// TwinCAT 3 PLC project PeerToPeerB
// ProgramVersion: 3.1.0.5
// libraries:
//   Tc2_Standard, * (Beckhoff Automation GmbH)
//   Tc2_System, * (Beckhoff Automation GmbH)
//   Tc2_TcpIp, * (Beckhoff Automation GmbH)
//   Tc2_Utilities, * (Beckhoff Automation GmbH)
//   Tc3_Module, * (Beckhoff Automation GmbH)
// project tree:
//   Data types/ E_ClientServerSteps.TcDUT, ST_FrameFifoEntry.TcDUT
//   Global Variables/ Global_Variables.TcGVL
//   POUs/ FB_PeerToPeer.TcPOU, MAIN.TcPOU
//   POUs/Helper POUs/ FB_FrameFifo.TcPOU, FB_LogFifo.TcPOU
//   / StandardB.TcTTO
// real-time tasks:
//   TASK StandardB: cycle T#10ms, priority 21, ADS port 351

CONFIGURATION PeerToPeerB
    RESOURCE PLC ON TwinCAT3
        TASK StandardB(INTERVAL := T#10ms, PRIORITY := 21);
        PROGRAM MAIN WITH StandardB : MAIN;
    END_RESOURCE
END_CONFIGURATION

// ---- Data types/E_ClientServerSteps.TcDUT
TYPE E_ClientServerSteps :
(
	eUDP_STATE_IDLE		:= 0,
	eUDP_STATE_CREATE_START,
	eUDP_STATE_CREATE_WAIT,
	eUDP_STATE_SEND_START,
	eUDP_STATE_SEND_WAIT,
	eUDP_STATE_RECEIVE_START,
	eUDP_STATE_RECEIVE_WAIT,
	eUDP_STATE_CLOSE_START,
	eUDP_STATE_CLOSE_WAIT,
	eUDP_STATE_ERROR
);
END_TYPE

// ---- Data types/ST_FrameFifoEntry.TcDUT
TYPE ST_FrameFifoEntry :
STRUCT
	stRemoteAddr 	: ST_SockAddr;(* Remote address. String containing an (Ipv4) Internet Protocol dotted address and port number. *)
	sMessage		: T_MaxString;	(* UDP packet data *)
END_STRUCT
END_TYPE

// ---- Global Variables/Global_Variables.TcGVL
VAR_GLOBAL CONSTANT
	PLCPRJ_BUFFER_SIZE					: UDINT := 1000;(* Max. internal fifo/receiver buffer size *)

	(* Some project specific error codes *)
	PLCPRJ_ERROR_SENDFIFO_OVERFLOW		: UDINT := 16#8103;
	PLCPRJ_ERROR_RECFIFO_OVERFLOW		: UDINT := 16#8104;
END_VAR

// ---- POUs/MAIN.TcPOU
PROGRAM MAIN
VAR
	bSendOnceToItself	: BOOL;(* Rising edge at this variable sends message to local host/port (itself) *)
	bSendOnceToRemote	: BOOL;(* Rising edge at this variable sends message to the remote host/port *)
	sSrvNetId			: T_AmsNetID 	:= '';(* TwinCAT TCP/IP server network address. Default: empty string. *)
	sLocalHost			: T_IPv4Addr 	:= '127.0.0.1';(* Local address: String containing an (Ipv4) Internet Protocol dotted address. *) 
	nLocalPort			: UDINT			:= 11000;(* Local address: IP port number *)
	sRemoteHost			: T_IPv4Addr 	:= '127.0.0.1';(* Remote address: String containing an (Ipv4) Internet Protocol dotted address. *)
	nRemotePort			: UDINT 		:= 10000;(* Remote address: IP port number. *)
	bEnable				: BOOL 			:= TRUE;(* TRUE => Enable/connect, FALSE => Disable/disconnect *)
	bLog				: BOOL			:= TRUE;(* TRUE => Enable log message output, FALSE => Disable *)
	
	fbPeerToPeer		: FB_PeerToPeer := ( sPrefix := 'PeerToPeerB::' ) ;
	
   	fbTx				: FB_FrameFifo;
   	fbRx				: FB_FrameFifo;
   	fbLog				: FB_LogFifo;
	
   	stSendTo			: ST_FrameFifoEntry;
   	stReceivedFrom		: ST_FrameFifoEntry;
	sLoggedMessage		: T_MaxString;

   	fbCloseAll 			: FB_SocketCloseAll;
   	bInitialize			: BOOL := TRUE;
END_VAR

(* On PLC reset or program download close all opened/created sockets *)
fbCloseAll( sSrvNetId := sSrvNetId, bExecute:= bInitialize );
IF fbCloseAll.bBusy OR fbCloseAll.bError THEN
	RETURN;
END_IF
bInitialize := FALSE;

(* Send and receive messages *)
fbPeerToPeer( 	sSrvNetId := sSrvNetId, 
				fbTx := fbTx, 
				fbRx := fbRx,
				fbLog := fbLog, 
				sLocalHost := sLocalHost, 
				nLocalPort := nLocalPort, 
				bEnable := bEnable, bLog := bLog );

IF fbPeerToPeer.bCreated THEN
	
	IF bSendOnceToRemote THEN
		bSendOnceToRemote 			:= FALSE;		(* Clear flag *)
		stSendTo.stRemoteAddr.sAddr := sRemoteHost;	(* Remote host IP address *)
		stSendTo.stRemoteAddr.nPort := nRemotePort;	(* Remote host port number *)
		stSendTo.sMessage			:= 'Hello remote host!';(* Message text *)
		fbTx.AddTail( stPut := stSendTo );	(* Add new entry to the send queue *)
		IF NOT fbTx.bOk THEN				(* Check for fifo overflow *)
			fbLog.Error( sMessage := 'FB_FrameFifo(sender)', nErrID := PLCPRJ_ERROR_SENDFIFO_OVERFLOW );
		END_IF
	END_IF
	
	IF bSendOnceToItself THEN
		bSendOnceToItself 			:= FALSE;		(* Clear flag *)
		stSendTo.stRemoteAddr.sAddr := sLocalHost;	(* Remote host == sLocalHost =>send it to itself *)
		stSendTo.stRemoteAddr.nPort := nLocalPort;	(* Remote port == nLocalPort => send it to itself *)
		stSendTo.sMessage			:= 'Hello itself!';(* Message text *)
		fbTx.AddTail( stPut := stSendTo );	(* Add new entry to the send queue *)
		IF NOT fbTx.bOk THEN				(* Check for fifo overflow *)
			fbLog.Error( sMessage := 'FB_FrameFifo(sender)', nErrID := PLCPRJ_ERROR_SENDFIFO_OVERFLOW );
		END_IF
	END_IF
	
END_IF
				
(* Remove all received frames from queue *)
REPEAT
	fbRx.RemoveHead( );
	IF fbRx.bOk THEN

		(* TODO:: Implement received frame handler *)
		stReceivedFrom := fbRx.stGet;
(*		ADSLOGSTR( ADSLOG_MSGTYPE_HINT OR ADSLOG_MSGTYPE_LOG OR ADSLOG_MSGTYPE_MSGBOX, '%s', stReceivedFrom.sMessage ); *)
		
	END_IF
UNTIL NOT fbRx.bOk
END_REPEAT

(* Remove all log messages from queue *)
REPEAT
	fbLog.Remove( );
	IF fbLog.bOk THEN

		(* TODO:: Implement log message handler *)
		sLoggedMessage := fbLog.sGet;

	END_IF
UNTIL NOT fbLog.bOk
END_REPEAT

END_PROGRAM

// ---- POUs/FB_PeerToPeer.TcPOU
(* Function block example of UDP peer-to-peer application *)
FUNCTION_BLOCK FB_PeerToPeer
VAR_IN_OUT
	fbTx		: FB_FrameFifo;(* TX fifo *)
	fbRx		: FB_FrameFifo;(* RX fifo *)
	fbLog		: FB_LogFifo;(* Log message fifo *)
END_VAR
VAR_INPUT
	sSrvNetId		: T_AmsNetID 	:= '';(* TwinCAT TCP/IP server network address. Default: empty string. *)
	sLocalHost		: T_IPv4Addr 	:= '127.0.0.1';(* Local address: String containing an (Ipv4) Internet Protocol dotted address. *)
	nLocalPort		: UDINT 		:= 0;(* Local address: IP port number. *)
	bEnable 		: BOOL			:= FALSE;(* TRUE => Enable/connect, FALSE => Disable/disconnect *)
	tReconnect		: TIME			:= T#5S;(* Reconnect delay time *)
	bLog			: BOOL			:= FALSE;(* TRUE => Enable log message output, FALSE => Disable *)
	sPrefix			: STRING 		:= 'PeerToPeerX::';(* Log message description string (allows the identification of log message source) *)
END_VAR
VAR_OUTPUT
	bCreated		: BOOL;(* Connectionless socket state (TRUE => created, FALSE => closed) *)
END_VAR
VAR
	fbCreate		: FB_SocketUdpCreate;
	fbClose			: FB_SocketClose;
	fbReceiveFrom	: FB_SocketUdpReceiveFrom;
	fbSendTo		: FB_SocketUdpSendTo;
	stSendTo		: ST_FrameFifoEntry;
	stReceivedFrom	: ST_FrameFifoEntry;
	fbCreateTimer	: TON := ( PT := T#0S );	
	eStep			: E_ClientServerSteps;
END_VAR

CASE eStep OF
	eUDP_STATE_IDLE:
		IF bEnable XOR bCreated THEN
			IF bEnable THEN
				fbTx.Clear( sPrefix := CONCAT( sPrefix, 'FB_FrameFifo(sender)::' ), bLog := bLog );(* Clear send fifo *)
				fbRx.Clear( sPrefix := CONCAT( sPrefix, 'FB_FrameFifo(receiver)::' ), bLog := bLog );(* Clear receiver fifo *)
				fbLog.Clear( sPrefix := sPrefix, bLog := bLog );(* Clear log fifo *)

				(* At program start (first time) connect emmediately, next time after delay time *)
				fbCreateTimer( IN := TRUE );
				IF fbCreateTimer.Q THEN
					fbCreateTimer( IN := FALSE, PT := tReconnect ); 
					eStep := eUDP_STATE_CREATE_START;
				END_IF
			ELSE
				eStep := eUDP_STATE_CLOSE_START;
			END_IF
		ELSIF bCreated THEN
			fbTx.RemoveHead( stGet => stSendTo );
			IF fbTx.bOk THEN
				eStep := eUDP_STATE_SEND_START;
			ELSE (* Empty *)
				eStep := eUDP_STATE_RECEIVE_START;
			END_IF
		ELSE
			fbCreateTimer( IN := FALSE, PT := T#0S );
		END_IF

	eUDP_STATE_CREATE_START:
		fbCreate( bExecute := FALSE  );
		fbCreate( sSrvNetId := sSrvNetId, sLocalHost:= sLocalHost, nLocalPort:= nLocalPort, bExecute:= TRUE );
		eStep := eUDP_STATE_CREATE_WAIT;

	eUDP_STATE_CREATE_WAIT:
		fbCreate( bExecute := FALSE );
		IF NOT fbCreate.bBusy THEN
			IF NOT fbCreate.bError THEN
				bCreated := TRUE;
				fbLog.Message( sMessage := 'Connectionless (UDP) socket created!', hSocket := fbCreate.hSocket );
				eStep := eUDP_STATE_IDLE;
			ELSE
				fbLog.Error( sMessage := 'FB_SocketUdpCreate()', nErrID := fbCreate.nErrID );
				eStep := eUDP_STATE_ERROR;
			END_IF
		END_IF

	eUDP_STATE_SEND_START:
		fbSendTo( bExecute := FALSE );
		fbSendTo( sSrvNetId := sSrvNetId, sRemoteHost := stSendTo.stRemoteAddr.sAddr,
					nRemotePort := stSendTo.stRemoteAddr.nPort,
					pSrc:= ADR( stSendTo.sMessage ),
					cbLen:= INT_TO_UDINT(LEN( stSendTo.sMessage )) + 1, (* Include the end delimiter *)
					hSocket:= fbCreate.hSocket, bExecute:= TRUE );
		eStep := eUDP_STATE_SEND_WAIT;

	eUDP_STATE_SEND_WAIT:
		fbSendTo( bExecute := FALSE );
		IF NOT fbSendTo.bBusy THEN
			IF NOT fbSendTo.bError THEN
				eStep := eUDP_STATE_RECEIVE_START;
			ELSE
				fbLog.Error( sMessage := 'FB_SocketUdpSendTo()', nErrID := fbSendTo.nErrID );
				eStep := eUDP_STATE_ERROR;
			END_IF
		END_IF

	eUDP_STATE_RECEIVE_START:
		MEMSET( ADR( stReceivedFrom ), 0, SIZEOF( stReceivedFrom ) );
		fbReceiveFrom( bExecute := FALSE );
		fbReceiveFrom( sSrvNetId := sSrvNetId, 
						pDest:= ADR( stReceivedFrom.sMessage ),
						cbLen:= SIZEOF( stReceivedFrom.sMessage ) - 1, (* Without string delimiter *)
						hSocket:= fbCreate.hSocket, bExecute:= TRUE );
		eStep := eUDP_STATE_RECEIVE_WAIT;

	eUDP_STATE_RECEIVE_WAIT:
		fbReceiveFrom( bExecute := FALSE );
		IF NOT fbReceiveFrom.bBusy THEN
			IF NOT fbReceiveFrom.bError THEN
				IF fbReceiveFrom.nRecBytes > 0 THEN
					
					stReceivedFrom.stRemoteAddr.sAddr := fbReceiveFrom.sRemoteHost;
					stReceivedFrom.stRemoteAddr.nPort := fbReceiveFrom.nRemotePort;
					
					fbRx.AddTail( stPut := stReceivedFrom );
					IF NOT fbRx.bOk THEN(* Check for fifo overflow *)
						fbLog.Error( sMessage :='FB_FrameFifo(receiver)', nErrID := PLCPRJ_ERROR_RECFIFO_OVERFLOW );
					END_IF
				END_IF
				eStep := eUDP_STATE_IDLE;
			ELSE
				fbLog.Error( sMessage := 'FB_SocketUdpReceiveFrom()', nErrID := fbReceiveFrom.nErrID );
				IF fbReceiveFrom.nErrID = 16#80072746 THEN(* Connection is reset by remote side *)
					eStep := eUDP_STATE_IDLE;
				ELSE
					eStep := eUDP_STATE_ERROR;
				END_IF
			END_IF
		END_IF

	eUDP_STATE_CLOSE_START:
		fbLog.Message( sMessage := 'Closing connectionless (UDP) socket!', hSocket := fbCreate.hSocket );
		fbClose( bExecute := FALSE );
		fbClose( sSrvNetId := sSrvNetId, hSocket := fbCreate.hSocket, bExecute := TRUE );
		eStep := eUDP_STATE_CLOSE_WAIT;

	eUDP_STATE_CLOSE_WAIT:
		fbClose( bExecute := FALSE );
		IF NOT fbClose.bBusy THEN
			bCreated := FALSE;
			IF NOT fbClose.bError THEN
				eStep := eUDP_STATE_IDLE;
			ELSE
				fbLog.Error( sMessage := 'FB_SocketClose()', nErrID := fbClose.nErrID );
				eStep := eUDP_STATE_ERROR;
			END_IF
		END_IF

	eUDP_STATE_ERROR: (* Error step *)
		IF bCreated THEN
			eStep := eUDP_STATE_CLOSE_START;
		ELSE
			eStep := eUDP_STATE_IDLE;
		END_IF
END_CASE

END_FUNCTION_BLOCK

// ---- POUs/Helper POUs/FB_FrameFifo.TcPOU
(* Tx/Rx (string data) fifo control function block *)
FUNCTION_BLOCK FB_FrameFifo
VAR_INPUT
	bLog		: BOOL := FALSE;(* TRUE => Enable log message output, FALSE => Disable *)
	sPrefix		: STRING := 'Unknown::';(* Log message description string (allows the identification of log message source) *)
	stPut		: ST_FrameFifoEntry;(* Frame entry to add (write) to the buffer *)
END_VAR
VAR_OUTPUT
	bOk			: BOOL;(* TRUE = New entry added or removed succesfully, FALSE = Fifo overflow or fifo empty *)
	stGet		: ST_FrameFifoEntry;(* Frame entry removed (read) from fifo *)
	nCount		: UDINT := 0;(* Number of fifo entries *)
END_VAR
VAR
	fbBuffer 	: FB_MemRingBuffer;(* Basic (lower level) string buffer control function block *)
	buffer		: ARRAY[0..PLCPRJ_BUFFER_SIZE] OF BYTE;(* Internal buffer memory *)
END_VAR

;

ACTION RemoveHead:
(* Removes oldest fifo entry *)
IF nCount = 0 THEN
	stGet.sMessage := '';
	stGet.stRemoteAddr.nPort := 0;
	stGet.stRemoteAddr.sAddr := '';
	bOk := FALSE;
	RETURN;
END_IF

fbBuffer.A_RemoveHead( pBuffer:= ADR(buffer), cbBuffer:= SIZEOF(buffer),
						pRead := ADR( stGet ), cbRead := SIZEOF( stGet ),
						bOk=>bOk, nCount=>nCount );
END_ACTION

ACTION Clear:
(* Clears all fifo entries *)
stGet.sMessage := '';
stGet.stRemoteAddr.nPort := 0;
stGet.stRemoteAddr.sAddr := '';
fbBuffer.A_Reset( pBuffer := ADR( buffer ), cbBuffer := SIZEOF( buffer ), 
					bOk=>bOk, nCount=>nCount );
END_ACTION

ACTION AddTail:
(* Adds new fifo entry *)
fbBuffer.A_AddTail( pBuffer:= ADR(buffer), cbBuffer:= SIZEOF(buffer),
					pWrite:= ADR( stPut ), cbWrite := SIZEOF( stPut ), 
					bOk=>bOk, nCount=>nCount );
IF bOk AND bLog THEN(* Log message *)
	ADSLOGSTR( ADSLOG_MSGTYPE_HINT OR ADSLOG_MSGTYPE_LOG, 
			CONCAT( CONCAT( sPrefix, SOCKETADDR_TO_STRING(stPut.stRemoteAddr) ), '>>"%s"' ),
			stPut.sMessage );
END_IF
END_ACTION

END_FUNCTION_BLOCK

// ---- POUs/Helper POUs/FB_LogFifo.TcPOU
(* Log/debug/error message fifo *)
FUNCTION_BLOCK FB_LogFifo
VAR_INPUT
	bLog		: BOOL 		:= FALSE;(* TRUE => Enable log message output, FALSE => Disable *)
	sPrefix		: STRING 	:= 'Unknown::';(* Log message description string (allows the identification of log message source) *)
	
	sMessage	: STRING 	:= '';(* String message to add (write) to the fifo *)
	nErrID		: UDINT 	:= 0;(* Error code to add (write) to the fifo *)
	hSocket		: T_HSOCKET;(* Socket connection handle *)
END_VAR
VAR_OUTPUT
	bOk			: BOOL;(* TRUE = New entry added or removed succesfully, FALSE = Fifo overflow or fifo empty *)
	sGet		: T_MaxString := '';(* String entry removed (read) from fifo *)
	nCount		: UDINT := 0;(* Number of fifo entries *)
END_VAR
VAR
	fbBuffer 	: FB_StringRingBuffer;(* Basic (lower level) string buffer control function block *)
	buffer		: ARRAY[0..PLCPRJ_BUFFER_SIZE] OF BYTE;(* Internal buffer memory *)
	sSource		: T_MaxString;	
	sPut		: T_MaxString;
END_VAR

;

ACTION Clear:
(* Clears all fifo entries *)
fbBuffer.A_Reset( 	pBuffer := ADR( buffer ), cbBuffer := SIZEOF( buffer ), 
					bOk=>bOk, nCount=>nCount, getValue=>sGet );
END_ACTION

ACTION Error:
(* Adds new fifo entry *)
IF nErrID = 0 THEN
	sSource := '::Error: 0x';
ELSIF ( nErrID AND 16#80000000) = 16#80000000 THEN
	IF nErrID = 16#80072746 THEN
		sSource := '::Win32 error (the connection is reset by remote side): 0x';
	ELSE
		sSource := '::Win32 error: 0x';
	END_IF
ELSIF (nErrID AND 16#00008100) = 16#00008100 THEN
	CASE nErrID OF
		PLCPRJ_ERROR_SENDFIFO_OVERFLOW:
			sSource := '::PLC sample project send fifo overflow error: 0x';
		PLCPRJ_ERROR_RECFIFO_OVERFLOW:
			sSource := '::PLC sample project receive fifo overflow error: 0x';
	ELSE
		sSource := '::Other PLC sample project error: 0x';
	END_CASE
ELSIF (nErrID AND 16#00008000) = 16#00008000 THEN
	sSource := '::Internal TCP/IP Connection Server error: 0x';
ELSE
	sSource := '::TwinCAT System error: 0x';
END_IF

sPut := CONCAT( CONCAT( CONCAT( sPrefix, sMessage ), sSource ), DWORD_TO_HEXSTR( nErrID AND 16#FFFF, 0, FALSE ) ); 

fbBuffer.A_AddTail( pBuffer:= ADR(buffer), cbBuffer:= SIZEOF(buffer),
					putValue:= sPut, bOk=>bOk, nCount=>nCount );
IF bOk THEN
	IF bLog THEN(* Log error message *)
		ADSLOGSTR( ADSLOG_MSGTYPE_ERROR OR ADSLOG_MSGTYPE_LOG, '%s', sPut );	
	END_IF
END_IF
END_ACTION

ACTION Remove:
(* Removes oldest fifo entry *)
IF nCount = 0 THEN
	sGet := '';
	bOk := FALSE;
	RETURN;
END_IF

fbBuffer.A_RemoveHead( pBuffer:= ADR(buffer), cbBuffer:= SIZEOF(buffer),
						getValue=>sGet, bOk=>bOk, nCount=>nCount );
END_ACTION

ACTION Message:
(* Adds new fifo entry *)
sPut := CONCAT( CONCAT( sPrefix, sMessage ), CONCAT( '::', SOCKETADDR_TO_STRING(hSocket.localAddr) ) );
fbBuffer.A_AddTail( pBuffer:= ADR(buffer), cbBuffer:= SIZEOF(buffer),
					putValue:= sPut, bOk=>bOk, nCount=>nCount );
IF bOk THEN
	IF bLog THEN(* Log information message *)
		ADSLOGSTR( ADSLOG_MSGTYPE_HINT OR ADSLOG_MSGTYPE_LOG, '%s', sPut );	
	END_IF
END_IF
END_ACTION

END_FUNCTION_BLOCK
